FUNCTION_BLOCK Slider (* Composite Function Block Type *)
  (* Standard: 61499-2 *)
  (* Version 0.0, 5/26/2016, Andrei, nxtControl GmbH, template *)
  PACKAGE Main;
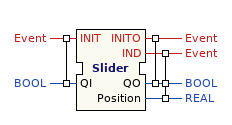
  EVENT_INPUT
    INIT WITH QI; (* Initialization Request *)
  END_EVENT
  EVENT_OUTPUT
    INITO WITH QO; (* Initialization Confirm *)
    IND WITH QO, Position; (* Execution Confirmation *)
  END_EVENT
  VAR_INPUT
    QI : BOOL; (* Input event qualifier *)
  END_VAR
  VAR_OUTPUT
    QO : BOOL; (* Output event qualifier *)
    Position : REAL;
  END_VAR
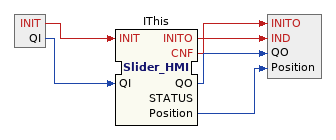
  FBS
    IThis : Slider_HMI;
  END_FBS
  EVENT_CONNECTIONS
    INIT TO IThis.INIT;
    IThis.INITO TO INITO;
    IThis.CNF TO IND;
  END_CONNECTIONS
  DATA_CONNECTIONS
    QI TO IThis.QI;
    IThis.QO TO QO;
    IThis.Position TO Position;
  END_CONNECTIONS
END_FUNCTION_BLOCK
